// Mitsubishi GX Works2 project: PLCQ_20-06   PLC: Q02/Q02H

PROGRAM MAIN
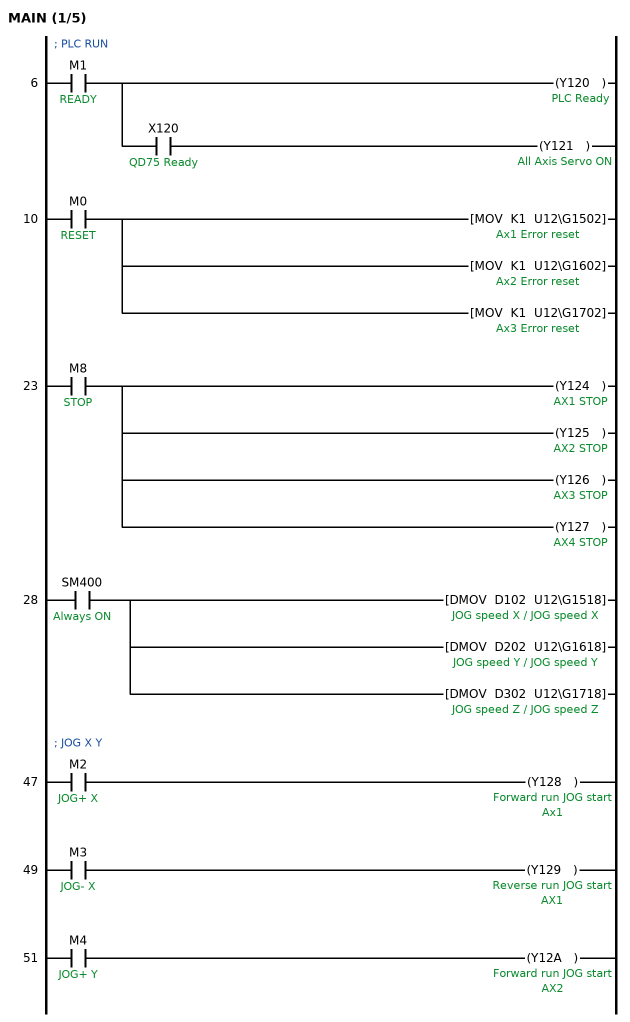
; PLC RUN
6     LD      M1  ; READY
      OUT     Y120  ; PLC Ready
      AND     X120  ; QD75 Ready
      OUT     Y121  ; All Axis Servo ON
10    LD      M0  ; RESET
      MOV     K1 U12\G1502  ; Ax1 Error reset
      MOV     K1 U12\G1602  ; Ax2 Error reset
      MOV     K1 U12\G1702  ; Ax3 Error reset
23    LD      M8  ; STOP
      OUT     Y124  ; AX1 STOP
      OUT     Y125  ; AX2 STOP
      OUT     Y126  ; AX3 STOP
      OUT     Y127  ; AX4 STOP
28    LD      SM400  ; Always ON
      DMOV    D102 U12\G1518  ; JOG speed X / JOG speed X
      DMOV    D202 U12\G1618  ; JOG speed Y / JOG speed Y
      DMOV    D302 U12\G1718  ; JOG speed Z / JOG speed Z
; JOG X Y
47    LD      M2  ; JOG+ X
      OUT     Y128  ; Forward run JOG start Ax1
49    LD      M3  ; JOG- X
      OUT     Y129  ; Reverse run JOG start AX1
51    LD      M4  ; JOG+ Y
      OUT     Y12A  ; Forward run JOG start AX2
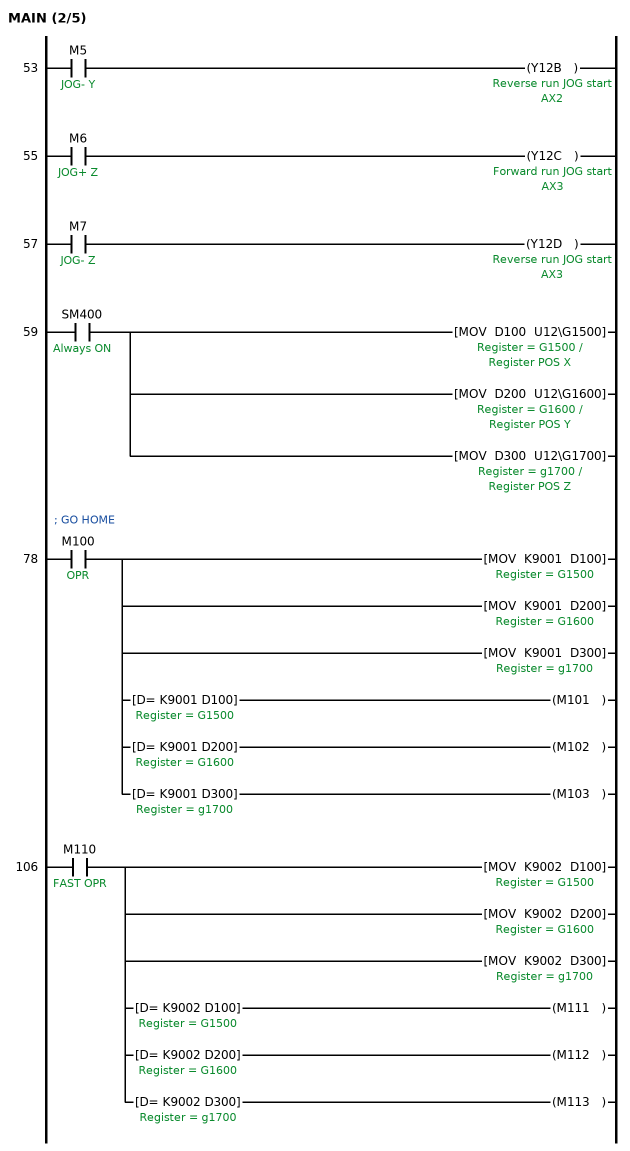
53    LD      M5  ; JOG- Y
      OUT     Y12B  ; Reverse run JOG start AX2
55    LD      M6  ; JOG+ Z
      OUT     Y12C  ; Forward run JOG start AX3
57    LD      M7  ; JOG- Z
      OUT     Y12D  ; Reverse run JOG start AX3
59    LD      SM400  ; Always ON
      MOV     D100 U12\G1500  ; Register = G1500 / Register POS X
      MOV     D200 U12\G1600  ; Register = G1600 / Register POS Y
      MOV     D300 U12\G1700  ; Register = g1700 / Register POS Z
; GO HOME
78    LD      M100  ; OPR
      MOV     K9001 D100
      MOV     K9001 D200
      MOV     K9001 D300
      MPS
      ANDD=   K9001 D100  ; Register = G1500
      OUT     M101
      MRD
      ANDD=   K9001 D200  ; Register = G1600
      OUT     M102
      MPP
      ANDD=   K9001 D300  ; Register = g1700
      OUT     M103
106   LD      M110  ; FAST OPR
      MOV     K9002 D100
      MOV     K9002 D200
      MOV     K9002 D300
      MPS
      ANDD=   K9002 D100  ; Register = G1500
      OUT     M111
      MRD
      ANDD=   K9002 D200  ; Register = G1600
      OUT     M112
      MPP
      ANDD=   K9002 D300  ; Register = g1700
      OUT     M113
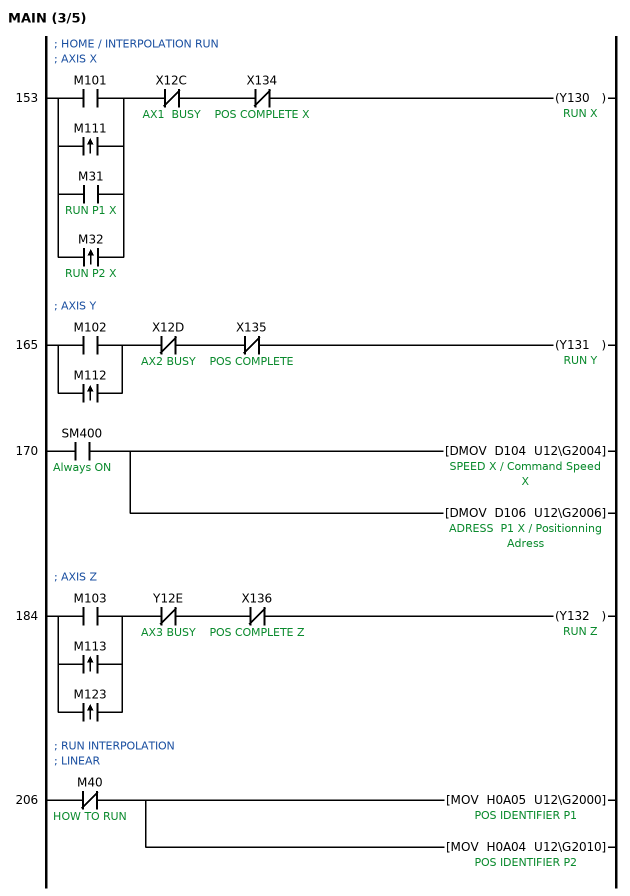
; HOME / INTERPOLATION RUN
; AXIS X
153   LD      M101
      ORP     M111
      OR      M31  ; RUN P1 X
      ORP     M32  ; RUN P2 X
      ANI     X12C  ; AX1  BUSY
      ANI     X134  ; POS COMPLETE X
      OUT     Y130  ; RUN X
; AXIS Y
165   LD      M102
      ORP     M112
      ANI     X12D  ; AX2 BUSY
      ANI     X135  ; POS COMPLETE
      OUT     Y131  ; RUN Y
170   LD      SM400  ; Always ON
      DMOV    D104 U12\G2004  ; SPEED X / Command Speed X
      DMOV    D106 U12\G2006  ; ADRESS  P1 X / Positionning Adress
; AXIS Z
184   LD      M103
      ORP     M113
      ORP     M123
      ANI     Y12E  ; AX3 BUSY
      ANI     X136  ; POS COMPLETE Z
      OUT     Y132  ; RUN Z
; RUN INTERPOLATION
; LINEAR
206   LDI     M40  ; HOW TO RUN
      MOV     H0A05 U12\G2000  ; POS IDENTIFIER P1
      MOV     H0A04 U12\G2010  ; POS IDENTIFIER P2
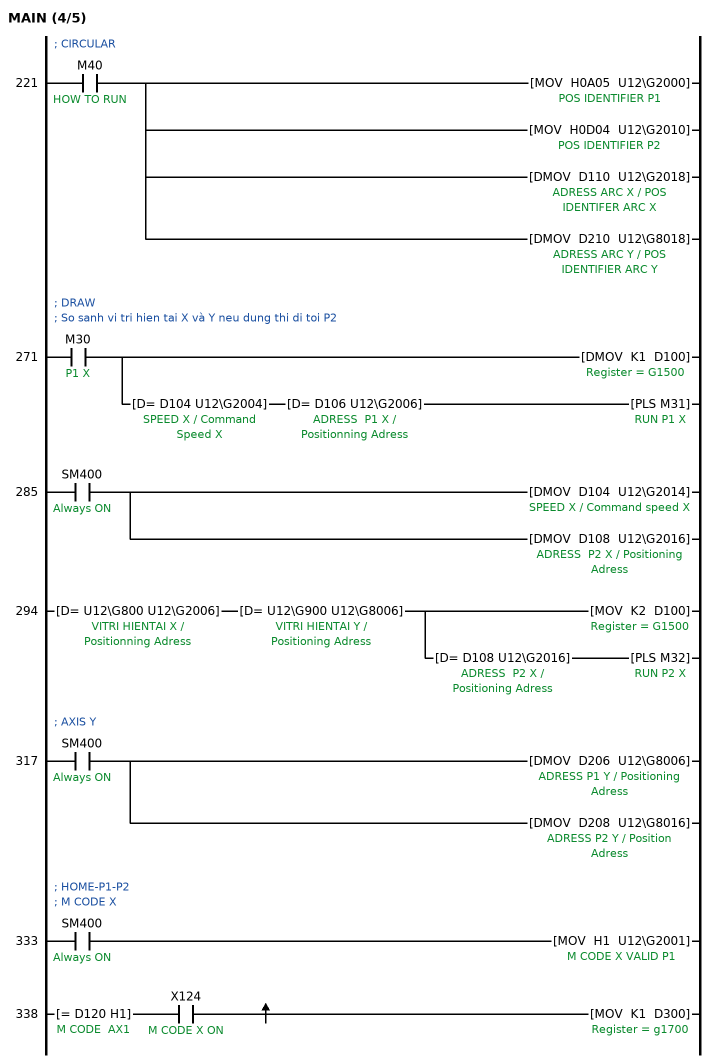
; CIRCULAR
221   LD      M40  ; HOW TO RUN
      MOV     H0A05 U12\G2000
      MOV     H0D04 U12\G2010
      DMOV    D110 U12\G2018  ; ADRESS ARC X / POS IDENTIFER ARC X
      DMOV    D210 U12\G8018  ; ADRESS ARC Y / POS IDENTIFIER ARC Y
; DRAW
; So sanh vi tri hien tai X và Y neu dung thi di toi P2
271   LD      M30  ; P1 X
      DMOV    K1 D100
      ANDD=   D104 U12\G2004  ; SPEED X / Command Speed X
      ANDD=   D106 U12\G2006  ; ADRESS  P1 X / Positionning Adress
      PLS     M31  ; RUN P1 X
285   LD      SM400  ; Always ON
      DMOV    D104 U12\G2014  ; Command speed X
      DMOV    D108 U12\G2016  ; ADRESS  P2 X / Positioning Adress
294   LDD=    U12\G800 U12\G2006  ; VITRI HIENTAI X / Positionning Adress
      ANDD=   U12\G900 U12\G8006  ; VITRI HIENTAI Y / Positioning Adress
      MOV     K2 D100
      ANDD=   D108 U12\G2016  ; ADRESS  P2 X / Positioning Adress
      PLS     M32  ; RUN P2 X
; AXIS Y
317   LD      SM400  ; Always ON
      DMOV    D206 U12\G8006  ; ADRESS P1 Y
      DMOV    D208 U12\G8016  ; ADRESS P2 Y / Position Adress
; HOME-P1-P2
; M CODE X
333   LD      SM400  ; Always ON
      MOV     H1 U12\G2001  ; M CODE X VALID P1
338   LD=     D120 H1  ; M CODE  AX1
      AND     X124  ; M CODE X ON
      MEP
      MOV     K1 D300
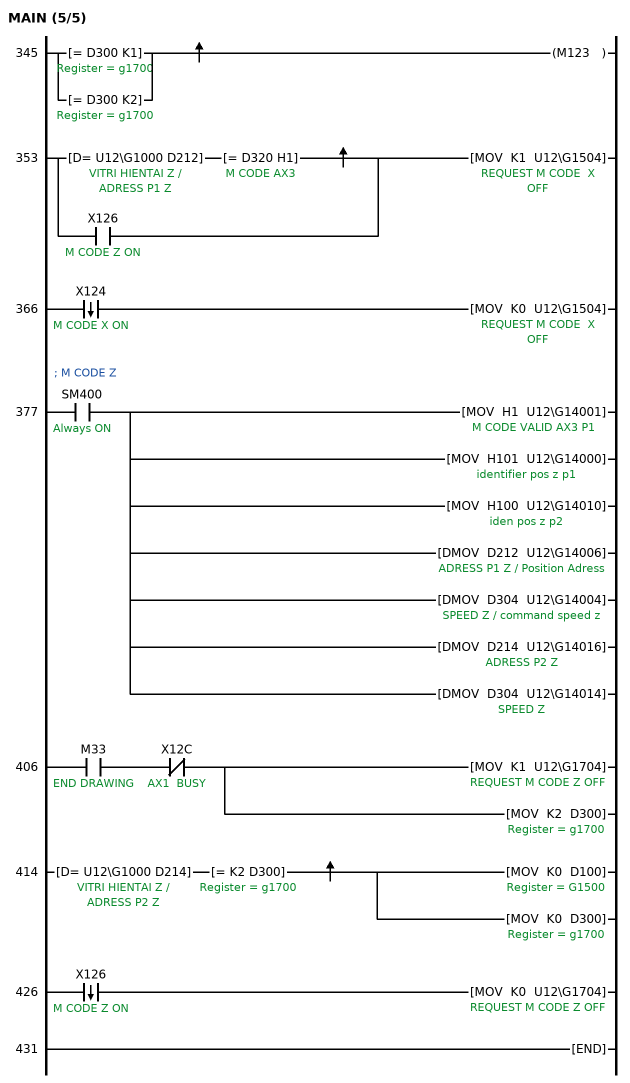
345   LD=     D300 K1  ; Register = g1700
      OR=     D300 K2  ; Register = g1700
      MEP
      OUT     M123
353   LDD=    U12\G1000 D212  ; VITRI HIENTAI Z / ADRESS P1 Z
      AND=    D320 H1  ; M CODE AX3
      MEP
      OR      X126  ; M CODE Z ON
      MOV     K1 U12\G1504  ; REQUEST M CODE  X OFF
366   LDF     X124  ; M CODE X ON
      MOV     K0 U12\G1504
; M CODE Z
377   LD      SM400  ; Always ON
      MOV     H1 U12\G14001  ; M CODE VALID AX3 P1
      MOV     H101 U12\G14000  ; identifier pos z p1
      MOV     H100 U12\G14010  ; iden pos z p2
      DMOV    D212 U12\G14006  ; Position Adress
      DMOV    D304 U12\G14004  ; SPEED Z / command speed z
      DMOV    D214 U12\G14016  ; ADRESS P2 Z
      DMOV    D304 U12\G14014
406   LD      M33  ; END DRAWING
      ANI     X12C  ; AX1  BUSY
      MOV     K1 U12\G1704  ; REQUEST M CODE Z OFF
      MOV     K2 D300
414   LDD=    U12\G1000 D214  ; VITRI HIENTAI Z / ADRESS P2 Z
      AND=    K2 D300  ; Register = g1700
      MEP
      MOV     K0 D100
      MOV     K0 D300
426   LDF     X126  ; M CODE Z ON
      MOV     K0 U12\G1704
431   END
END_PROGRAM

// device comments not shown above
X50  ; QD75 READY
Y50  ; PLC READY
Y58  ; JOG+
Y59  ; JOG-
M20  ; SET HOME X
M21  ; RETURN HOME X
M22  ; HOME X
D0  ; Speed
D1  ; JOG SPEED
D204  ; SPEED Y
